PROGRAM MAIN
VAR_INPUT
	Controlword AT%Q*		: UINT;	
	TargetPosition AT%Q*	: DINT;
END_VAR
VAR_OUTPUT
	Statusword AT%I*		: UINT;
END_VAR

VAR
	bStartUpTest			: BOOL;
	bVelocityModeActive		: BOOL := FALSE;
END_VAR	

VAR
	aTemperatureObjects		: ARRAY[1..2] OF INT := [1,1]; 	//0x2200, 0x2202
	aMOPObjects				: ARRAY[1..2] OF INT := [1,1]; 	//0x6060, 0x6061
	aControlStatusWords		: ARRAY[1..2] OF INT := [1,1]; 	//0x6040, 0x6041
	bTargetPosition			: BOOL;							//0x607A
	
	fbSetToPPMode			: FB_EcCoeSdoWrite;
	fbSetToVelocityMode		: FB_EcCoeSdoWrite;
	bSetToPPMode			: BOOL;
	bSetToVelocityMode		: BOOL;// := TRUE;
	tSetToPPMode			: TON;
	fSetToVelocityMode		: F_TRIG;
	nModeOfOperation		: UDINT := 2;
	bBasicTest 				: BOOL := FALSE;
END_VAR

//StartUpTests(bTrigger := bStartUpTest,
//	aTemperatureObjects := aTemperatureObjects,
//	aControlStatusWords := aControlStatusWords,
//	aMOPObjects := aMOPObjects,
//	sNetID := GVL.sNetId,
//	nSlaveAddr := GVL.nSlaveAddr);
(*
fbSetToPPMode(sNetId := GVL.sNetId, 
				nSlaveAddr := GVL.nSlaveAddr,
				nIndex := 16#6060,
				pSrcBuf := ADR(nModeOfOperation),
				cbBufLen := SIZEOF (nModeOfOperation),
				bExecute := bSetToPPMode);
tSetToPPMode(IN := bSetToPPMode,
				PT := T#250MS);
bSetToPPMode := TRUE;
IF tSetToPPMode.Q THEN
	P_ProfilePositionModeTest();	
END_IF
*)
IF bBasicTest THEN
	BasicTests();
ELSE
//TODO read IF velocitymode was set via FB
fbSetToVelocityMode(sNetId := GVL.sNetId, 
				nSlaveAddr := GVL.nSlaveAddr,
				nIndex := 16#6060,
				pSrcBuf := ADR(nModeOfOperation),
				cbBufLen := SIZEOF (nModeOfOperation),
				bExecute := bSetToVelocityMode);
fSetToVelocityMode(CLK := fbSetToVelocityMode.bBusy);

IF fSetToVelocityMode.Q THEN
	bVelocityModeActive := TRUE;
	ADSLOGSTR(msgCtrlMask := ADSLOG_MSGTYPE_HINT,
				msgFmtStr := 'Set to velocity mode.',
				strArg := '');
END_IF
IF bVelocityModeActive THEN
	P_VelocityModeTest();
END_IF
END_IF

END_PROGRAM

(* stored: Version 1.1.0.1, ProductVersion 3.1.4024.11
   POU MAIN: Id {adcae204-ece0-4dbd-83bc-e75c85ce708f}, SpecialFunc None *)
